INTERFACE ITF_TopElement1_HMI_Init EXTENDS ITF_BaseTopElement, ITF_TopElement1_HMI_Lacznik

END_INTERFACE

(* stored: Version 1.1.0.1, ProductVersion 3.1.4024.15
   Itf ITF_TopElement1_HMI_Init: Id {d0ab8372-f443-0c59-18c3-2fd0f26fb4a6} *)
